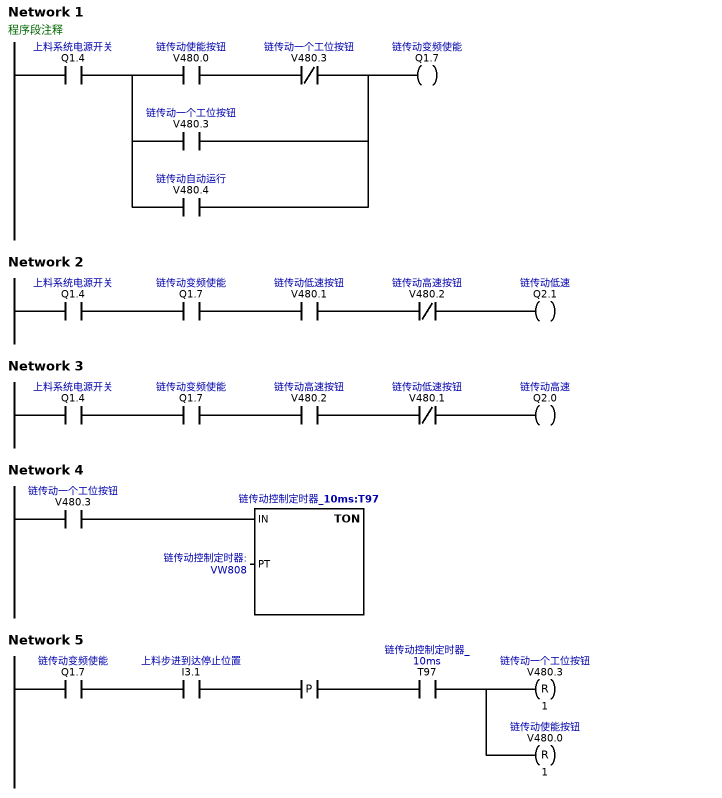
[picture p24: SBR19 networks 1-5]
Network 1
// 程序段注释
LD     上料系统电源开关:Q1.4
LD     链传动使能按钮:V480.0
AN     链传动一个工位按钮:V480.3
O      链传动一个工位按钮:V480.3
O      链传动自动运行:V480.4
ALD
=      链传动变频使能:Q1.7
Network 2
LD     上料系统电源开关:Q1.4
A      链传动变频使能:Q1.7
A      链传动低速按钮:V480.1
AN     链传动高速按钮:V480.2
=      链传动低速:Q2.1
Network 3
LD     上料系统电源开关:Q1.4
A      链传动变频使能:Q1.7
A      链传动高速按钮:V480.2
AN     链传动低速按钮:V480.1
=      链传动高速:Q2.0
Network 4
LD     链传动一个工位按钮:V480.3
TON    链传动控制定时器_10ms:T97, 链传动控制定时器:VW808
Network 5
LD     链传动变频使能:Q1.7
A      上料步进到达停止位置:I3.1
EU
A      链传动控制定时器_10ms:T97
R      链传动一个工位按钮:V480.3, 1
R      链传动使能按钮:V480.0, 1
END_SUBROUTINE_BLOCK

SUBROUTINE_BLOCK 数据初始化:SBR20
TITLE=子程序注释
BEGIN
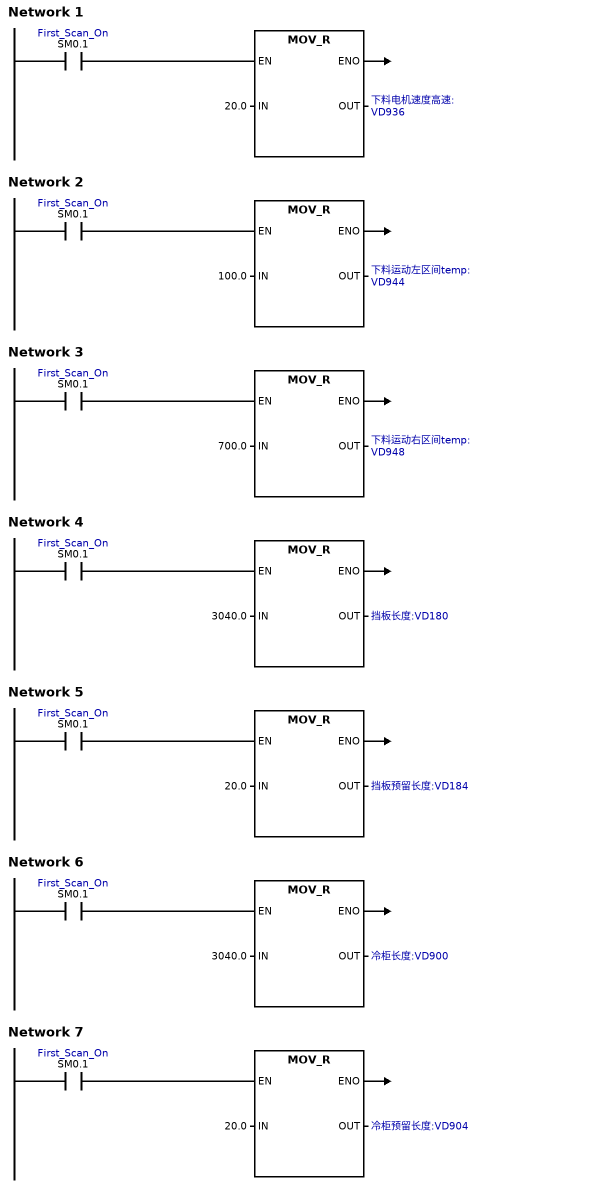
Network 1
LD     First_Scan_On:SM0.1
MOVR   20.0, 下料电机速度高速:VD936
Network 2
LD     First_Scan_On:SM0.1
MOVR   100.0, 下料运动左区间temp:VD944
Network 3
LD     First_Scan_On:SM0.1
MOVR   700.0, 下料运动右区间temp:VD948
Network 4
LD     First_Scan_On:SM0.1
MOVR   3040.0, 挡板长度:VD180
Network 5
LD     First_Scan_On:SM0.1
MOVR   20.0, 挡板预留长度:VD184
Network 6
LD     First_Scan_On:SM0.1
MOVR   3040.0, 冷柜长度:VD900
Network 7
LD     First_Scan_On:SM0.1
MOVR   20.0, 冷柜预留长度:VD904
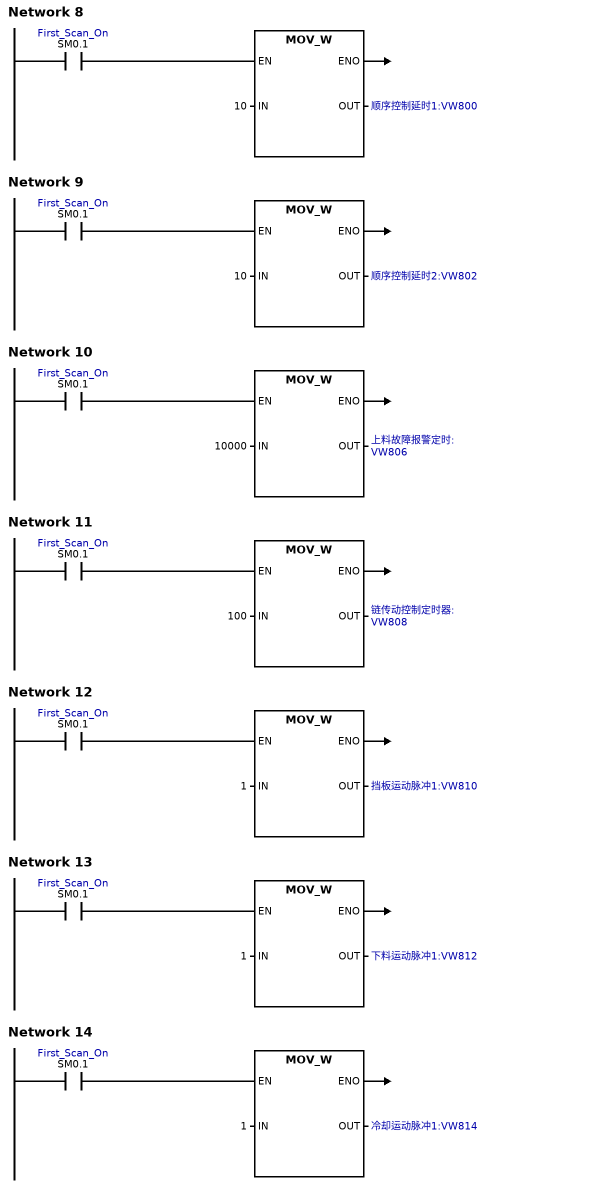
Network 8
LD     First_Scan_On:SM0.1
MOVW   10, 顺序控制延时1:VW800
Network 9
LD     First_Scan_On:SM0.1
MOVW   10, 顺序控制延时2:VW802
Network 10
LD     First_Scan_On:SM0.1
MOVW   10000, 上料故障报警定时:VW806
Network 11
LD     First_Scan_On:SM0.1
MOVW   100, 链传动控制定时器:VW808
Network 12
LD     First_Scan_On:SM0.1
MOVW   1, 挡板运动脉冲1:VW810
Network 13
LD     First_Scan_On:SM0.1
MOVW   1, 下料运动脉冲1:VW812
Network 14
LD     First_Scan_On:SM0.1
MOVW   1, 冷却运动脉冲1:VW814
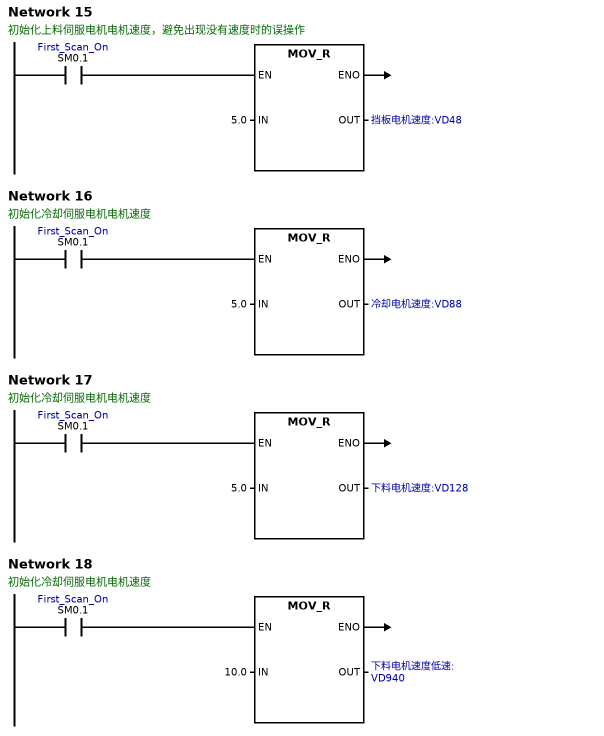
Network 15
// 初始化上料伺服电机电机速度，避免出现没有速度时的误操作
LD     First_Scan_On:SM0.1
MOVR   5.0, 挡板电机速度:VD48
Network 16
// 初始化冷却伺服电机电机速度
LD     First_Scan_On:SM0.1
MOVR   5.0, 冷却电机速度:VD88
Network 17
// 初始化冷却伺服电机电机速度
LD     First_Scan_On:SM0.1
MOVR   5.0, 下料电机速度:VD128
Network 18
// 初始化冷却伺服电机电机速度
LD     First_Scan_On:SM0.1
MOVR   10.0, 下料电机速度低速:VD940
END_SUBROUTINE_BLOCK

SUBROUTINE_BLOCK 故障报警:SBR21
TITLE=子程序注释
BEGIN
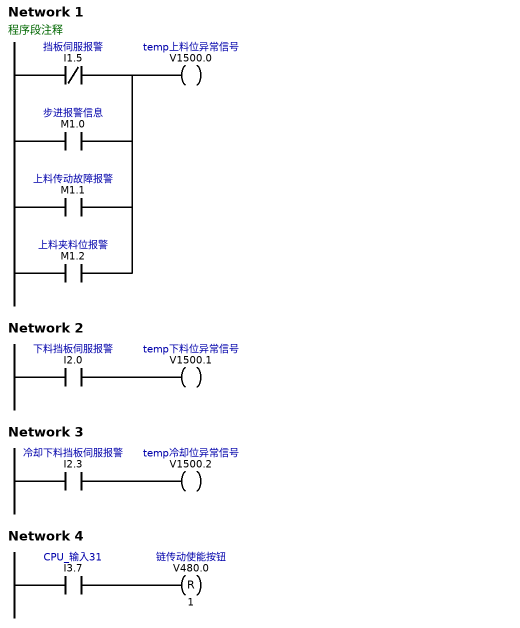
Network 1
// 程序段注释
LDN    挡板伺服报警:I1.5
O      步进报警信息:M1.0
O      上料传动故障报警:M1.1
O      上料夹料位报警:M1.2
=      temp上料位异常信号:V1500.0
Network 2
LD     下料挡板伺服报警:I2.0
=      temp下料位异常信号:V1500.1
Network 3
LD     冷却下料挡板伺服报警:I2.3
=      temp冷却位异常信号:V1500.2
Network 4
LD     CPU_输入31:I3.7
R      链传动使能按钮:V480.0, 1
END_SUBROUTINE_BLOCK
